TYPE T_MODBUS_CFG EXTENDS T_RS_COMM_CFG:
STRUCT
END_STRUCT
END_TYPE

(* stored: Version 1.1.0.1, ProductVersion 3.1.4022.16
   DUT T_MODBUS_CFG: Id {0397cdf9-4e21-4e69-9691-8a8d415fbcb9} *)
